Universal Robots PolyScope program: Short_PHomeToInvB.urp

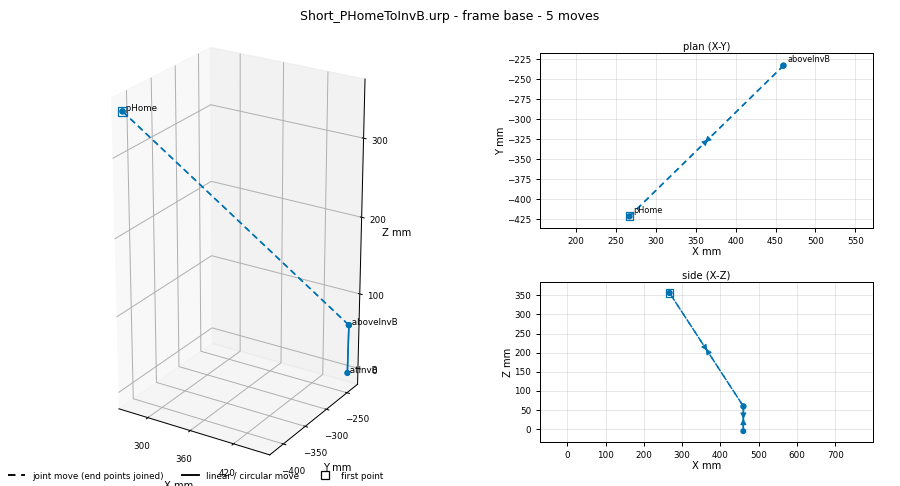
[picture p0: tool path of Short_PHomeToInvB.urp in frame base, 5 of 5 moves have a stored position in this frame; points joined in program order, loops and branches not executed]
Program Short_PHomeToInvB (installation=admin directory=/programs/THU_530PM/Final createdIn=3.8.0.61336 lastSavedIn=3.15.8.106339 robotSerialNumber=2015350924)
Calibrated DH parameters: a=[0, -0.425, -0.39225, 0, 0, 0]; d=[0.089159, 0, 0, 0.10915, 0.09465, 0.0823]; alpha=[1.570796, 0, 0, 1.570796, -1.570796, 0]; deltaTheta=[0, 0, 0, 0, 0, 0]
Robot Program (runOnlyOnce=true)
  Call _adminLinearIndex2
  MoveJ speed 180 deg/s, acceleration 200 deg/s^2 (useActiveTCP=true)
    Waypoint pHome: TCP in base x=267.143 y=-421.455 z=355.857 mm, rx=1.114 ry=1.106 rz=0.0051 rad; joints [-44.997, -90.001, -89.999, -90.001, 90.004, 0.008] deg; flange x=267.141 y=-421.459 z=431.857 mm, rx=-1.2021 ry=2.9025 rz=0.0001 rad
    Waypoint aboveInvB: motionParameters(blendRadius=0.048); TCP in base x=460.044 y=-232.62 z=59.707 mm, rx=1.706 ry=-0.0085 rz=-1.2116 rad; joints [-14.573, -107.855, -116.733, -45.605, 89.915, 120.716] deg; flange x=460.32 y=-232.575 z=135.707 mm, rx=-1.2083 ry=-2.8965 rz=0.003 rad
  MoveL speed 15 mm/s, acceleration 15 mm/s^2 (useActiveTCP=true) feature=Base
    Waypoint atInvB: TCP in base x=459.62 y=-233.005 z=-4.986 mm, rx=1.706 ry=-0.0084 rz=-1.2116 rad; joints [-14.628, -115.357, -119.202, -35.638, 89.916, 120.661] deg; flange x=459.901 y=-232.963 z=71.013 mm, rx=-1.2083 ry=-2.8965 rz=0.003 rad
    Set DigitalOutput pin=digital_out[0]; digitalValue=0
    Wait Sleep waitTime=1
    Waypoint aboveInvB: motionParameters(blendRadius=0.05); TCP in base x=460.044 y=-232.62 z=59.707 mm, rx=1.706 ry=-0.0085 rz=-1.2116 rad; joints [-14.573, -107.855, -116.733, -45.605, 89.915, 120.716] deg; flange x=460.32 y=-232.575 z=135.707 mm, rx=-1.2083 ry=-2.8965 rz=0.003 rad
  MoveJ speed 90 deg/s, acceleration 100 deg/s^2 (useActiveTCP=true)
    Waypoint pHome: TCP in base x=267.143 y=-421.455 z=355.857 mm, rx=1.114 ry=1.106 rz=0.0051 rad; joints [-44.997, -90.001, -89.999, -90.001, 90.004, 0.008] deg; flange x=267.141 y=-421.459 z=431.857 mm, rx=-1.2021 ry=2.9025 rz=0.0001 rad
SubProgram  [hidden by the author, left out]
SubProgram _adminLinearIndex2 [hidden by the author, left out]
